// TIA Portal V19 export
TYPE "LAF_typeJobs"
TITLE = LAF_typeJob
// Job data
// stored: Access Published
   STRUCT
      enableManualCtrl { ExternalWritable := 'False'} : Bool;   // Jobs can be controlled via hmiInterface
      commands : "LAF_typeJobsCommands";
      status { ExternalWritable := 'False'} : "LAF_typeJobsStatus";   // Control of the job management
      previousJobs { ExternalWritable := 'False'} : Array[0..63] of "LAF_typeJobPrevious";   // List of the previous jobs
   END_STRUCT;
END_TYPE
